Staubli VAL3: clkValve14.pgx

program clkValve14()
begin
  call toggleValve(14)
end
